(* CoDeSys 2.3 export: ALARMFIRE.EXP *)

(* POU _БИБЛИОТЕКИ/Alarms/AlarmFire, CFC *)
FUNCTION_BLOCK	AlarmFire	(*	ФБ фиксации аварии пожара	*)
VAR_INPUT
	TrackingOn	: BOOL;	(*	Условие отслеживания аварии (True - отслеживать, False - не отслеживать)	*)
	Status			: BOOL;	(*	Статус сигнала	*)
	TypeContact	: BOOL := FALSE;	(*	Тип контатка статуса (False - NC, True - NO)	*)
	Delay			: REAL;	(*	Задержка срабатывания аварии, сек	*)
	Reset			: BOOL;	(*	Сброс аварии	*)
END_VAR
VAR_OUTPUT
	Alarm			: BOOL;	(*	Авария!	*)
END_VAR
VAR
	DelayTon		: TON;	(*	Таймер задержки срабатывания аварии	*)
END_VAR
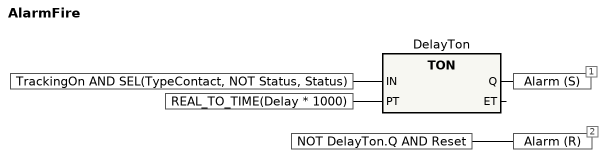
_CFC_ (* Continuous Function Chart, elements in execution order *)
#0 DelayTon:TON(IN: TrackingOn AND SEL(TypeContact, NOT Status, Status), PT: REAL_TO_TIME(Delay * 1000))
#1 S Alarm <= #0.Q
#2 R Alarm <= NOT DelayTon.Q AND Reset
_END_CFC_
(* the same logic as Structured Text *)
DelayTon(IN := TrackingOn AND SEL(TypeContact, NOT Status, Status), PT := REAL_TO_TIME(Delay * 1000));
IF DelayTon.Q THEN Alarm := TRUE; END_IF;
IF NOT DelayTon.Q AND Reset THEN Alarm := FALSE; END_IF;
END_FUNCTION_BLOCK
